Universal Robots PolyScope program: align_peg.urp

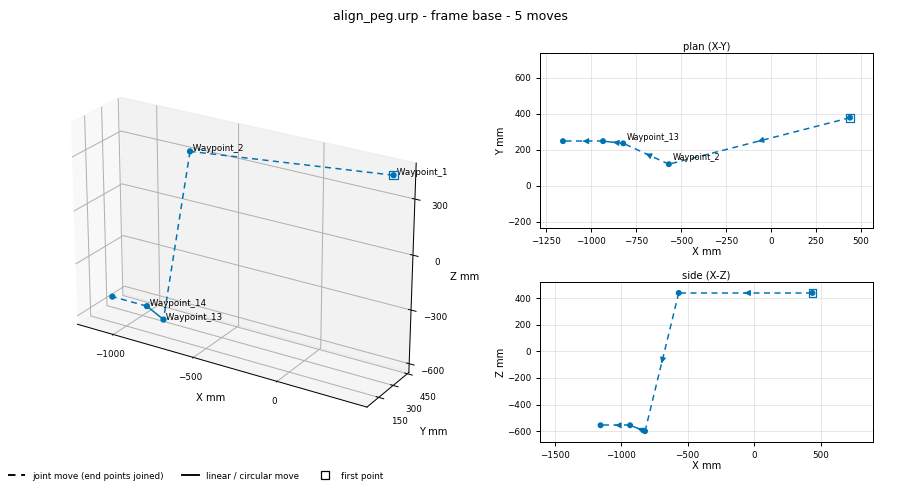
[picture p0: tool path of align_peg.urp in frame base, 5 of 5 moves have a stored position in this frame; points joined in program order, loops and branches not executed]
Program align_peg (installation=default directory=/programs createdIn=5.21.3 lastSavedIn=5.21.3 robotSerialNumber=20246801938)
Calibrated DH parameters: a=[-0.000071, -0.790281, -0.600694, 0.000061, -0.000039, 0]; d=[0.236272, 604.465945, 132.116513, -736.382239, 0.159268, 0.154005]; alpha=[1.570254, -0.000567, 0.000559, 1.571709, -1.56999, 0]; deltaTheta=[0, -0.409357, 7.293326, -0.600784, -0.000001, -0.000001]
InitVariablesNode
Robot Program (runOnlyOnce=true)
  'leave home'
  SuppressedNode
    Set NoAction tcp=pretend_welder
  URCap MachineLogic for Universal Robots (MachineLogic for Universal Robots, Vention Inc.) dataModel(type=addMotor, numberAdded=0, speed_in_mm_per_min=3000.0, acceleration_in_mm_per_s2=50.0, ActuatorPos=750.0, teachColor=BLUE, combo1=MachineMotion1, combo2=(1) Custom Actuator, combo3=Move to Position, combo6=In series, message=Move to Position, description=Moves the actuator to a specified position from the home location., comboAddress=Address 1, comboActuator=Valve 1)
  SuppressedNode
    MoveJ speed 60 deg/s, acceleration 80 deg/s^2 (useActiveTCP=true optimoveEnabled=false optiMoveSpeed=0.3 optiMoveAcceleration=0.09) feature=Base
      Waypoint Waypoint_1: TCP in base x=439.488 y=377.651 z=439.882 mm, rx=2.2965 ry=2.0951 rz=-0.0644 rad; joints [-188.975, -96.657, 133.035, 103.058, 4.742, -139.298] deg; TCP offset x=-9.5 y=-328 z=105 mm, rx=1.2092 ry=-1.2092 rz=1.2092 rad
      Waypoint Waypoint_2: TCP in base x=-567.049 y=119.272 z=439.882 mm, rx=-0.8568 ry=2.9689 rz=0.0164 rad; joints [-61.526, -96.657, 133.035, 103.058, 4.742, -139.298] deg
  'spin?'
  'points'
  SuppressedNode
    If 1≟2
      'tilt'
      MoveJ speed 60 deg/s, acceleration 80 deg/s^2 (useActiveTCP=true optimoveEnabled=false optiMoveSpeed=0.3 optiMoveAcceleration=0.09) feature=Base
        Waypoint Waypoint_3: TCP in base x=-782.323 y=119.272 z=439.882 mm, rx=-0.1409 ry=-2.6543 rz=-0.0579 rad; joints [-38.432, -118.572, 138.524, -52.025, 61.559, 15.606] deg
        Waypoint Waypoint_4: TCP in base x=-839.555 y=157.82 z=59.483 mm, rx=-0.1359 ry=-2.576 rz=-0.0621 rad; joints [-38.672, -71.334, 157.907, -123.561, 62.634, 17.978] deg
      MoveJ speed 60 deg/s, acceleration 80 deg/s^2 (useActiveTCP=true optimoveEnabled=false optiMoveSpeed=0.3 optiMoveAcceleration=0.09) feature=Base
        Waypoint Waypoint_5: TCP in base x=-839.555 y=157.82 z=154.033 mm, rx=-0.1359 ry=-2.576 rz=-0.0621 rad; joints [-38.663, -86.736, 154.954, -105.21, 62.654, 17.987] deg
        Waypoint Waypoint_6: TCP in base x=-930.504 y=247.449 z=154.033 mm, rx=1.7264 ry=-2.0251 rz=0.4813 rad; joints [-47.448, -44.223, 108.584, -199.171, 48.598, 145.286] deg
        Waypoint Waypoint_7: TCP in base x=-1008.947 y=181.992 z=154.033 mm, rx=2.8737 ry=-0.4936 rz=0.8267 rad; joints [-21.503, -27.525, 68.369, -188.611, 91.899, 180.193] deg
        Waypoint Waypoint_8: TCP in base x=-1005.76 y=182.333 z=166.844 mm, rx=2.9972 ry=-0.3869 rz=0.8133 rad; joints [-19.507, -27.075, 40.49, 16.635, -93.289, 5.373] deg
      MoveJ speed 60 deg/s, acceleration 80 deg/s^2 (useActiveTCP=true optimoveEnabled=false optiMoveSpeed=0.3 optiMoveAcceleration=0.09) feature=Base
        Waypoint Waypoint_9: TCP in base x=-1005.76 y=135.995 z=-301.87 mm, rx=-2.9509 ry=-0.1653 rz=-0.7853 rad; joints [-11.926, -9.754, 42.428, -1.512, -104.955, 12.357] deg
      'actual'
      MoveJ speed 60 deg/s, acceleration 80 deg/s^2 (useActiveTCP=true optimoveEnabled=false optiMoveSpeed=0.3 optiMoveAcceleration=0.09) feature=Base
        Waypoint Waypoint_13: TCP in base x=-820.615 y=235.067 z=-600.712 mm, rx=2.789 ry=-0.3984 rz=-1.1799 rad; joints [-36.349, -28.171, 124.415, -140.933, -100.235, -24.393] deg
        Waypoint Waypoint_12: TCP in base x=-1004.07 y=104.199 z=-600.712 mm, rx=-1.7423 ry=1.8799 rz=0.9101 rad; joints [-16.137, -21.262, 116.105, -178.633, -44.236, 66.954] deg
        Waypoint Waypoint_11: TCP in base x=-1004.07 y=251.363 z=-600.712 mm, rx=0.2287 ry=2.3379 rz=0.1546 rad; joints [-20.059, -11.78, 93.702, -217.985, -87.895, 163.36] deg
        Waypoint Waypoint_10: TCP in base x=-813.178 y=367.752 z=-600.712 mm, rx=1.8208 ry=1.595 rz=-0.5735 rad; joints [-36.866, -15.96, 106.588, -203.107, -131.508, 223.468] deg
  SuppressedNode
    If 1≟2
      Folder first try
        'worked pretty good. my 4 points were not a circle so it moved kind of wonky. but still spun'
        MoveJ speed 60 deg/s, acceleration 80 deg/s^2 (useActiveTCP=true optimoveEnabled=false optiMoveSpeed=0.3 optiMoveAcceleration=0.09) feature=Base
          Waypoint Waypoint_13: TCP in base x=-820.615 y=235.067 z=-600.712 mm, rx=2.789 ry=-0.3984 rz=-1.1799 rad; joints [-36.349, -28.171, 124.415, -140.933, -100.235, -24.393] deg
        MoveP speed 10 mm/s, acceleration 1200 mm/s^2 (blendRadius=0.025 useActiveTCP=true optimoveEnabled=false optiMoveSpeed=0.3 optiMoveAcceleration=0.09) feature=Base
          CircleMove (OrientationMode=FIXED)
            Waypoint Waypoint_12: TCP in base x=-1004.07 y=104.199 z=-600.712 mm, rx=-1.7423 ry=1.8799 rz=0.9101 rad; joints [-16.137, -21.262, 116.105, -178.633, -44.236, 66.954] deg
            Waypoint Waypoint_11: TCP in base x=-1004.07 y=251.363 z=-600.712 mm, rx=0.2287 ry=2.3379 rz=0.1546 rad; joints [-20.059, -11.78, 93.702, -217.985, -87.895, 163.36] deg
          CircleMove (OrientationMode=FIXED)
            Waypoint Waypoint_10: TCP in base x=-813.178 y=367.752 z=-600.712 mm, rx=1.8208 ry=1.595 rz=-0.5735 rad; joints [-36.866, -15.96, 106.588, -203.107, -131.508, 223.468] deg
            Waypoint Waypoint_13: TCP in base x=-820.615 y=235.067 z=-600.712 mm, rx=2.789 ry=-0.3984 rz=-1.1799 rad; joints [-36.349, -28.171, 124.415, -140.933, -100.235, -24.393] deg
  SuppressedNode
    Folder second try
      'worked pretty good. my 4 points were not a circle so it moved kind of wonky. but still spun'
      MoveJ speed 60 deg/s, acceleration 80 deg/s^2 (useActiveTCP=true optimoveEnabled=false optiMoveSpeed=0.3 optiMoveAcceleration=0.09) feature=Base
        Waypoint Waypoint_13: TCP in base x=-820.615 y=235.067 z=-600.712 mm, rx=2.789 ry=-0.3984 rz=-1.1799 rad; joints [-36.349, -28.171, 124.415, -140.933, -100.235, -24.393] deg
      MoveL speed 250 mm/s, acceleration 1200 mm/s^2 (useActiveTCP=true optimoveEnabled=false optiMoveSpeed=0.3 optiMoveAcceleration=0.09) feature=Base
        Waypoint Waypoint_14: TCP in base x=-933.006 y=247.304 z=-556.073 mm, rx=2.8803 ry=-0.0661 rz=-1.2302 rad; joints [-29.557, -31.673, 118.683, -136.217, -107.709, -21.437] deg
      MoveP speed 10 mm/s, acceleration 1200 mm/s^2 (blendRadius=0.025 useActiveTCP=true optimoveEnabled=false optiMoveSpeed=0.3 optiMoveAcceleration=0.09) feature=Base
        CircleMove (OrientationMode=FIXED)
          Waypoint ViaPoint_1: TCP in base x=-997.806 y=207.515 z=-556.073 mm, rx=-1.6876 ry=1.8024 rz=0.7466 rad; joints [-20.307, -26.743, 112.915, -161.612, -48.271, 66.703] deg
          Waypoint EndPoint_1: TCP in base x=-1049.868 y=270.629 z=-561.34 mm, rx=0.1326 ry=2.3308 rz=-0.0225 rad; joints [-23.206, -14.525, 91.047, -209.147, -79.208, 166.32] deg
        CircleMove (OrientationMode=FIXED)
          Waypoint ViaPoint_2: TCP in base x=-979.337 y=322.737 z=-561.34 mm, rx=1.8079 ry=1.682 rz=-0.747 rad; joints [-31.834, -18.679, 101.995, -196.68, -128.219, 232.931] deg
          Waypoint Waypoint_14: TCP in base x=-933.006 y=247.304 z=-556.073 mm, rx=2.8803 ry=-0.0661 rz=-1.2302 rad; joints [-29.557, -31.673, 118.683, -136.217, -107.709, -21.437] deg
        CircleMove (OrientationMode=FIXED)
          Waypoint ViaPoint_1: TCP in base x=-997.806 y=207.515 z=-556.073 mm, rx=-1.6876 ry=1.8024 rz=0.7466 rad; joints [-20.307, -26.743, 112.915, -161.612, -48.271, 66.703] deg
          Waypoint EndPoint_1: TCP in base x=-1049.868 y=270.629 z=-561.34 mm, rx=0.1326 ry=2.3308 rz=-0.0225 rad; joints [-23.206, -14.525, 91.047, -209.147, -79.208, 166.32] deg
  SuppressedNode
    Folder third try
      'worked pretty good. my 4 points were not a circle so it moved kind of wonky. but still spun'
      MoveJ speed 60 deg/s, acceleration 80 deg/s^2 (useActiveTCP=true optimoveEnabled=false optiMoveSpeed=0.3 optiMoveAcceleration=0.09) feature=Base
        Waypoint Waypoint_13: TCP in base x=-820.615 y=235.067 z=-600.712 mm, rx=2.789 ry=-0.3984 rz=-1.1799 rad; joints [-36.349, -28.171, 124.415, -140.933, -100.235, -24.393] deg
      MoveL speed 250 mm/s, acceleration 1200 mm/s^2 (useActiveTCP=true optimoveEnabled=false optiMoveSpeed=0.3 optiMoveAcceleration=0.09) feature=Base
        Waypoint Waypoint_14: TCP in base x=-933.006 y=247.304 z=-556.073 mm, rx=2.8803 ry=-0.0661 rz=-1.2302 rad; joints [-29.557, -31.673, 118.683, -136.217, -107.709, -21.437] deg
      MoveJ speed 60 deg/s, acceleration 80 deg/s^2 (useActiveTCP=true optimoveEnabled=false optiMoveSpeed=0.3 optiMoveAcceleration=0.09) feature=Base
        Waypoint Waypoint_15: TCP in base x=-1155.523 y=247.304 z=-556.073 mm, rx=0.1075 ry=2.332 rz=-0.0118 rad; joints [-20.182, -12.844, 81.619, -201.64, -80.424, -192.34] deg
      MoveL speed 250 mm/s, acceleration 1200 mm/s^2 (useActiveTCP=true optimoveEnabled=false optiMoveSpeed=0.3 optiMoveAcceleration=0.09) feature=Base
        Waypoint EndPoint_1: TCP in base x=-1049.868 y=270.629 z=-561.34 mm, rx=0.1326 ry=2.3308 rz=-0.0225 rad; joints [-23.206, -14.525, 91.047, -209.147, -79.208, 166.32] deg
      Wait Sleep waitTime=1
      MoveP speed 10 mm/s, acceleration 1200 mm/s^2 (blendRadius=0.025 useActiveTCP=true optimoveEnabled=false optiMoveSpeed=0.3 optiMoveAcceleration=0.09) feature=Base
        CircleMove (OrientationMode=FIXED)
          Waypoint ViaPoint_2: TCP in base x=-979.337 y=322.737 z=-561.34 mm, rx=1.8079 ry=1.682 rz=-0.747 rad; joints [-31.834, -18.679, 101.995, -196.68, -128.219, 232.931] deg
          Waypoint Waypoint_14: TCP in base x=-933.006 y=247.304 z=-556.073 mm, rx=2.8803 ry=-0.0661 rz=-1.2302 rad; joints [-29.557, -31.673, 118.683, -136.217, -107.709, -21.437] deg
        CircleMove (OrientationMode=FIXED)
          Waypoint ViaPoint_1: TCP in base x=-997.806 y=207.515 z=-556.073 mm, rx=-1.6876 ry=1.8024 rz=0.7466 rad; joints [-20.307, -26.743, 112.915, -161.612, -48.271, 66.703] deg
          Waypoint EndPoint_1: TCP in base x=-1049.868 y=270.629 z=-561.34 mm, rx=0.1326 ry=2.3308 rz=-0.0225 rad; joints [-23.206, -14.525, 91.047, -209.147, -79.208, 166.32] deg
        CircleMove (OrientationMode=FIXED)
          Waypoint ViaPoint_2: TCP in base x=-979.337 y=322.737 z=-561.34 mm, rx=1.8079 ry=1.682 rz=-0.747 rad; joints [-31.834, -18.679, 101.995, -196.68, -128.219, 232.931] deg
          Waypoint Waypoint_14: TCP in base x=-933.006 y=247.304 z=-556.073 mm, rx=2.8803 ry=-0.0661 rz=-1.2302 rad; joints [-29.557, -31.673, 118.683, -136.217, -107.709, -21.437] deg
  SuppressedNode
    Folder fourth (peg)
      'worked pretty good. my 4 points were not a circle so it moved kind of wonky. but still spun'
      MoveJ speed 60 deg/s, acceleration 80 deg/s^2 (useActiveTCP=true optimoveEnabled=false optiMoveSpeed=0.3 optiMoveAcceleration=0.09) feature=Base
        Waypoint Waypoint_13: TCP in base x=-820.615 y=235.067 z=-600.712 mm, rx=2.789 ry=-0.3984 rz=-1.1799 rad; joints [-36.349, -28.171, 124.415, -140.933, -100.235, -24.393] deg
      MoveL speed 250 mm/s, acceleration 1200 mm/s^2 (useActiveTCP=true optimoveEnabled=false optiMoveSpeed=0.3 optiMoveAcceleration=0.09) feature=Base
        Waypoint Waypoint_14: TCP in base x=-933.006 y=247.304 z=-556.073 mm, rx=2.8803 ry=-0.0661 rz=-1.2302 rad; joints [-29.557, -31.673, 118.683, -136.217, -107.709, -21.437] deg
      MoveJ speed 60 deg/s, acceleration 80 deg/s^2 (useActiveTCP=true optimoveEnabled=false optiMoveSpeed=0.3 optiMoveAcceleration=0.09) feature=Base
        Waypoint Waypoint_15: TCP in base x=-1155.523 y=247.304 z=-556.073 mm, rx=0.1075 ry=2.332 rz=-0.0118 rad; joints [-20.182, -12.844, 81.619, -201.64, -80.424, -192.34] deg
      MoveL speed 250 mm/s, acceleration 1200 mm/s^2 (useActiveTCP=true optimoveEnabled=false optiMoveSpeed=0.3 optiMoveAcceleration=0.09) feature=Base
        Waypoint Waypoint_17: TCP in base x=-941.011 y=247.304 z=-664.711 mm, rx=0.1107 ry=2.4446 rz=-0.0059 rad; joints [-25.301, -8.351, 98.215, -228.375, -75.252, -194.663] deg
        Waypoint Waypoint_16: TCP in base x=-941.011 y=247.304 z=-712.565 mm, rx=0.1107 ry=2.4446 rz=-0.0059 rad; joints [-25.303, -5.145, 95.455, -228.821, -75.25, -194.666] deg
      Wait Sleep waitTime=2
      MoveP speed 10 mm/s, acceleration 1200 mm/s^2 (blendRadius=0.025 useActiveTCP=true optimoveEnabled=false optiMoveSpeed=0.3 optiMoveAcceleration=0.09) feature=Base
        CircleMove (OrientationMode=FIXED)
          Waypoint ViaPoint_3: TCP in base x=-902.128 y=271.937 z=-712.565 mm, rx=1.8739 ry=1.7594 rz=-0.6531 rad; joints [-29.151, -8.204, 102.29, -210.895, -134.312, -127.809] deg
          Waypoint EndPoint_2: TCP in base x=-879.998 y=228.196 z=-712.565 mm, rx=-2.9313 ry=0.1903 rz=1.0627 rad; joints [-28.767, -21.46, 113.717, -133.842, -105.761, -15.36] deg
        CircleMove (OrientationMode=FIXED)
          Waypoint ViaPoint_4: TCP in base x=-916.094 y=204.675 z=-712.565 mm, rx=-1.7817 ry=1.8631 rz=0.6704 rad; joints [-24.822, -17.392, 113.115, -161.812, -44.424, 56.385] deg
          Waypoint Waypoint_16: TCP in base x=-941.011 y=247.304 z=-712.565 mm, rx=0.1107 ry=2.4446 rz=-0.0059 rad; joints [-25.303, -5.145, 95.455, -228.821, -75.25, -194.666] deg
        CircleMove (OrientationMode=FIXED)
          Waypoint ViaPoint_3: TCP in base x=-902.128 y=271.937 z=-712.565 mm, rx=1.8739 ry=1.7594 rz=-0.6531 rad; joints [-29.151, -8.204, 102.29, -210.895, -134.312, -127.809] deg
          Waypoint EndPoint_2: TCP in base x=-879.998 y=228.196 z=-712.565 mm, rx=-2.9313 ry=0.1903 rz=1.0627 rad; joints [-28.767, -21.46, 113.717, -133.842, -105.761, -15.36] deg
  Folder fifth (backofhole)
    'worked pretty good. my 4 points were not a circle so it moved kind of wonky. but still spun'
    Set NoAction tcp=backofhole
    MoveJ speed 60 deg/s, acceleration 80 deg/s^2 (useActiveTCP=true optimoveEnabled=false optiMoveSpeed=0.3 optiMoveAcceleration=0.09) feature=Base
      Waypoint Waypoint_1: TCP in base x=439.488 y=377.651 z=439.882 mm, rx=2.2965 ry=2.0951 rz=-0.0644 rad; joints [-188.975, -96.657, 133.035, 103.058, 4.742, -139.298] deg
      Waypoint Waypoint_2: TCP in base x=-567.049 y=119.272 z=439.882 mm, rx=-0.8568 ry=2.9689 rz=0.0164 rad; joints [-61.526, -96.657, 133.035, 103.058, 4.742, -139.298] deg
    MoveJ speed 60 deg/s, acceleration 80 deg/s^2 (useActiveTCP=true optimoveEnabled=false optiMoveSpeed=0.3 optiMoveAcceleration=0.09) feature=Base
      Waypoint Waypoint_13: TCP in base x=-820.615 y=235.067 z=-600.712 mm, rx=2.789 ry=-0.3984 rz=-1.1799 rad; joints [-36.349, -28.171, 124.415, -140.933, -100.235, -24.393] deg
    MoveL speed 250 mm/s, acceleration 1200 mm/s^2 (useActiveTCP=true optimoveEnabled=false optiMoveSpeed=0.3 optiMoveAcceleration=0.09) feature=Base
      Waypoint Waypoint_14: TCP in base x=-933.006 y=247.304 z=-556.073 mm, rx=2.8803 ry=-0.0661 rz=-1.2302 rad; joints [-29.557, -31.673, 118.683, -136.217, -107.709, -21.437] deg
    MoveJ speed 60 deg/s, acceleration 80 deg/s^2 (useActiveTCP=true optimoveEnabled=false optiMoveSpeed=0.3 optiMoveAcceleration=0.09) feature=Base
      Waypoint Waypoint_15: TCP in base x=-1155.523 y=247.304 z=-556.073 mm, rx=0.1075 ry=2.332 rz=-0.0118 rad; joints [-20.182, -12.844, 81.619, -201.64, -80.424, -192.34] deg
    'end of approach'
    SuppressedNode
      MoveL speed 250 mm/s, acceleration 1200 mm/s^2 (useActiveTCP=true optimoveEnabled=false optiMoveSpeed=0.3 optiMoveAcceleration=0.09) feature=Base
        Waypoint Waypoint_18: TCP in base x=-939.675 y=242.159 z=-688.931 mm, rx=0.1858 ry=2.4403 rz=-0.0331 rad; joints [-25.871, -6.691, 96.723, -229.022, -77.473, -192.661] deg; TCP offset x=4.51 y=-328 z=105 mm, rx=1.2092 ry=-1.2092 rz=1.2092 rad
        Waypoint Waypoint_19: TCP in base x=-939.675 y=242.159 z=-719.896 mm, rx=0.1858 ry=2.4403 rz=-0.0331 rad; joints [-25.872, -4.62, 94.895, -229.263, -77.472, -192.663] deg
    SuppressedNode
      Wait Sleep waitTime=2
    SuppressedNode
      MoveP speed 10 mm/s, acceleration 1200 mm/s^2 (blendRadius=0.025 useActiveTCP=true optimoveEnabled=false optiMoveSpeed=0.3 optiMoveAcceleration=0.09) feature=Base
        CircleMove (OrientationMode=FIXED)
          Waypoint ViaPoint_5: TCP in base x=-907.205 y=264.785 z=-719.9 mm, rx=1.8738 ry=1.7594 rz=-0.6531 rad; joints [-28.993, -7.691, 102.75, -211.731, -134.382, -127.614] deg
          Waypoint EndPoint_3: TCP in base x=-881.393 y=236.092 z=-719.9 mm, rx=-2.9216 ry=0.2235 rz=1.0597 rad; joints [-28.315, -21.001, 113.308, -133.575, -104.432, -14.143] deg
        CircleMove (OrientationMode=FIXED)
          Waypoint ViaPoint_6: TCP in base x=-912.548 y=210.58 z=-719.9 mm, rx=-1.7177 ry=1.9091 rz=0.6478 rad; joints [-24.877, -16.344, 111.718, -164.775, -43.133, 60.968] deg
          Waypoint Waypoint_19: TCP in base x=-939.675 y=242.159 z=-719.896 mm, rx=0.1858 ry=2.4403 rz=-0.0331 rad; joints [-25.872, -4.62, 94.895, -229.263, -77.472, -192.663] deg
        CircleMove (OrientationMode=FIXED)
          Waypoint ViaPoint_5: TCP in base x=-907.205 y=264.785 z=-719.9 mm, rx=1.8738 ry=1.7594 rz=-0.6531 rad; joints [-28.993, -7.691, 102.75, -211.731, -134.382, -127.614] deg
          Waypoint EndPoint_3: TCP in base x=-881.393 y=236.092 z=-719.9 mm, rx=-2.9216 ry=0.2235 rz=1.0597 rad; joints [-28.315, -21.001, 113.308, -133.575, -104.432, -14.143] deg
